FUNCTION_BLOCK DoubleCylinderBaseImplemented  EXTENDS TcoPneumatics.TcoDoubleCylinderBase

SUPER^(inoAtHomePos1 := inoAtHomePos1,inoAtHomePos2 := inoAtHomePos2, inoAtWorkPos1 := inoAtWorkPos1,inoAtWorkPos2 := inoAtWorkPos2, inoToHomePos := inoToHomePos, inoToWorkPos := inoToWorkPos);

PROPERTY MoveHomeTask : TcoCore.ITcoTask
GET
END_GET
SET
END_SET
END_PROPERTY

PROPERTY MoveWorkTask : TcoCore.ITcoTask
GET
END_GET
SET
END_SET
END_PROPERTY

PROPERTY StopTask : TcoCore.ITcoTask
GET
END_GET
SET
END_SET
END_PROPERTY

END_FUNCTION_BLOCK

(* stored: Version 1.1.0.1, ProductVersion 3.1.4024.10
   POU DoubleCylinderBaseImplemented: Id {96688d48-3e7e-0014-2727-2445de349ebf}, SpecialFunc None
   Property MoveHomeTask: Id {df688880-b7dd-080b-06e9-e459028a2fd8}
   Get Get: Id {8c28e51f-f44d-0626-3637-c3f7c8f251af}
   Set Set: Id {4e4f657a-f2c6-03cf-0c03-a7cce6b6f8f5}
   Property MoveWorkTask: Id {ba155310-480e-0131-112a-09529b0cf0d1}
   Get Get: Id {f92b3cdc-9ec0-09d8-025d-bf979f706c25}
   Set Set: Id {594a452f-f1fa-0992-0445-a40e42f2918a}
   Property StopTask: Id {1e2c12f6-1b4a-0ce7-3f10-ec75afe63456}
   Get Get: Id {044a8542-f139-0d2c-1579-57075c051b03}
   Set Set: Id {2d423797-dc04-08b9-0ab2-8e4de40450af} *)
